PROGRAM prg_Setpointsturing
VAR
	DrukPlus, DrukMin		AT		%I*		:BOOL;
	SetPoint		:INT:=0;
	LangerAls1sec: TON;
	LANGEPLUS: TON;
	LANGEMIN: TON;
	SetpointWaarde: REAL;
	KorteDrukPlus: F_TRIG;
	KorteDrukMin: F_TRIG;
	SpanningUit		AT			%Q*			:REAL;
END_VAR

LANGEPLUS(IN:= DrukPlus, PT:= T#1S);
LANGEMIN(IN:= DrukMin, PT:= T#1S);

SetpointWaarde := INT_TO_REAL (SetPoint) * 1000	/32767;

IF LANGEPLUS.Q THEN
	SetpointWaarde:= SetpointWaarde + 100;
ELSIF LANGEMIN.Q THEN
	SetpointWaarde:= SetpointWaarde - 100;
END_IF

KorteDrukPlus(CLK:= DrukPlus);
KorteDrukMin(CLK:= DrukMin);

IF KorteDrukPlus.Q AND NOT LANGEPLUS.Q THEN
	SetpointWaarde:= SetpointWaarde + 1;
ELSIF KorteDrukMin.Q AND NOT LANGEMIN.Q THEN
	SetpointWaarde:= SetpointWaarde - 1;
END_IF

SpanningUit:= SetpointWaarde / 100;

END_PROGRAM

(* stored: Version 1.1.0.1, ProductVersion 3.1.4024.15
   POU prg_Setpointsturing: Id {6a0f88b7-fb46-465c-8ecf-3f86cad7e03d}, SpecialFunc None *)
